{attribute 'qualified_only'}
{attribute 'strict'}
{attribute 'to_string'}
TYPE eRobMoveType :
(
	LinearToolSpace 			:= 0,		// Move to position (linear in tool-space)
	LinearJointSpace 			:= 1,		// Move to position (linear in joint-space)
	CircularToolSpace 			:= 2,		// Move Circular: Move to position (circular in tool-space)
	BlendCircularMoveLinear		:= 3		// Move Process
);
END_TYPE

(* stored: Version 1.1.0.1
   DUT eRobMoveType: Id {c64abdee-f51e-4995-84e5-9dcd86fa6fff} *)
